// TwinCAT 3 PLC project PLC
// ProgramVersion: 3.1.4024.0
// libraries:
//   Tc2_MC2, * (Beckhoff Automation GmbH)
//   Tc2_MC2_Drive, * (Beckhoff Automation GmbH)
//   Tc2_Standard, * (Beckhoff Automation GmbH)
//   Tc2_System, * (Beckhoff Automation GmbH)
//   Tc3_Module, * (Beckhoff Automation GmbH)
// project tree:
//   GVLs/ GVL.TcGVL
//   / PlcTask.TcTTO
//   POUs/ FB_AxisStMachine.TcPOU (not stored), FB_Axis.TcPOU, FB_AxisStMachineMaster.TcPOU, MAIN.TcPOU
// real-time tasks:
//   TASK PlcTask: cycle T#10ms, priority 20, ADS port 350
// motion (NC):
//   TASK NC-Task 1 SAF: cycle T#2ms, priority 4, ADS port 501
//   TASK NC-Task 1 SVB: cycle T#10ms, priority 8, ADS port 511
//   AXIS Stepper (id 1)
//     General: UnitName=°
//     Dynamic: Acceleration=4263.16, Deceleration=4263.16, Jerk=12789.5
//     Velo: RefSearch=28.42105, RefSync=28.42105, SlowManual=142.10525, FastManual=852.6315, Fast=2842.105, Maximum=2842.11
//     OtherSettings: AllowMotionCmdToSlave=true
//     encoder EncType=4
//       EncPara: ScaleFactorNumerator=360, ScaleFactorDenominator=4096, MaxCount=#x0000ffff
//         Inc: RefSoftSyncMask=#x0000ffff
//         TimeComp: EncDelayCycles=4
//     drive DrvType=24
//       Analog: VeloReferenz=7200, TorqueSetpointScale=10, ScaleFactorActTorque=0.1
//       TimeComp: TaskDelayCycles=1
//     controller CtrType=1
//       CtrPara: PriorControlFactor=1
//         PID: PosKp=50
//         Observer: BandWidth=20
//   AXIS Line1LeftA (id 2)
//     Dynamic: Acceleration=7354.05, Deceleration=7354.05, Jerk=22062.1
//     Velo: RefSearch=49.02699, RefSync=49.02699, SlowManual=245.13495, FastManual=1470.8097, Fast=4902.699, Maximum=4902.7
//     OtherSettings: AllowMotionCmdToSlave=true
//     encoder EncType=19
//       EncPara: ScaleFactorNumerator=60, ScaleFactorDenominator=1048576, MaxCount=#xffffffff
//     drive DrvType=16
//       DrvPara: MaxCount=#xffffffff, DriveControlDWord=#x00020100
//         Analog: VeloReferenz=5392.9689, VeloScale=71.5255737304688, TorqueSetpointScale=10, ScaleFactorActTorque=0.1
//         TimeComp: TaskDelayCycles=1
//     controller CtrType=1
//       CtrPara: PriorControlFactor=1
//         Observer: BandWidth=20
//   AXIS Line2RightB (id 3)
//     Dynamic: Acceleration=7354.05, Deceleration=7354.05, Jerk=22062.1
//     Velo: RefSearch=49.02699, RefSync=49.02699, SlowManual=245.13495, FastManual=1470.8097, Fast=4902.699, Maximum=4902.7
//     OtherSettings: AllowMotionCmdToSlave=true
//     encoder EncType=19
//       EncPara: ScaleFactorNumerator=60, ScaleFactorDenominator=1048576, MaxCount=#xffffffff
//     drive DrvType=16
//       DrvPara: MaxCount=#xffffffff, DriveControlDWord=#x00020100
//         Analog: VeloReferenz=5392.9689, VeloScale=71.5255737304688, TorqueSetpointScale=10, ScaleFactorActTorque=0.1
//         TimeComp: TaskDelayCycles=1
//     controller CtrType=1
//       CtrPara: PriorControlFactor=1
//         Observer: BandWidth=20
//   AXIS RobotMasterVirtualAxe (id 4)
//     OtherSettings: AllowMotionCmdToSlave=true
//     encoder EncType=1
//     drive DrvType=5
//       Analog: TorqueSetpointScale=10, ScaleFactorActTorque=0.1
//       TimeComp: TaskDelayCycles=1
//     controller CtrType=1
//       CtrPara: PriorControlFactor=1
//         Observer: BandWidth=20
// I/O:
//   DEVICE Device 2 (EtherCAT), AmsNetId 172.16.17.50.3.1
//     Term 1 (EK1100) [EK1100 EtherCAT Coupler (2A E-Bus)]
//       Term 2 (EL1004) [EL1004 4Ch. Dig. Input 24V, 3ms]
//       Term 3 (EL2004) [EL2004 4Ch. Dig. Output 24V, 0.5A]
//       Term 4 (EL3062) [EL3062 2Ch. Ana. Input 0-10V]
//       Term 5 (EL7037) [EL7037 1Ch. Stepper motor output stage (24V, 1.5A)]
//         startup 32786:5 := 02 // STM Features Ch.1 / Speed range
//         startup 32785:1 := DE01 // STM Controller Settings Ch.1 / Kp factor (curr.)
//         startup 32785:2 := A200 // STM Controller Settings Ch.1 / Ki factor (curr.)
//         startup 32788:3 := C0010000 // STM Controller Settings 3 Ch.1 / Kp factor (velo.)
//         startup 32788:4 := 8813 // STM Controller Settings 3 Ch.1 / Tn (velo.)
//         startup 32786:8 := 00 // STM Features Ch.1 / Feedback type
//       Term 6 (EL9510) [EL9510 Power supply terminal 10V]
//       Term 9 (EL9011) [EL9011 End Terminal]
//     Term 7 (AX8620-0000-0105) [AX8620-0000-0105]
//       Drive 8 (AX8206-0210-0104) [AX8206-0210-0104 (2Ch. 6A servo axis, safe-motion, multi-FB)]
//         modules: Device, Device, Device, Device, Device, Device, Device, Device, Device, Device, Device (Safety), Device, Device, Device, Device, Device, Device, Device, Device, Device, Device, Device, Device, Device, Device, Device, Device, Device, Device, Device, Device, Line1Left, Line1Left, Line1Left, Line1Left, Line1Left, Line1Left, Line1Left, Line1Left, Line1Left, Line1Left, Line1Left, Line1Left, Line1Left, Line1Left, Line1Left, Line1Left, Line1Left, Line1Left, Line1Left, Line1Left, Line1Left, Line1Left, Line1Left, Line1Left, Line1Left, Line1Left, Line2Right, Line2Right, Line2Right, Line2Right, Line2Right, Line2Right, Line2Right, Line2Right, Line2Right, Line2Right, Line2Right, Line2Right, Line2Right, Line2Right, Line2Right, Line2Right, Line2Right, Line2Right, Line2Right, Line2Right, Line2Right, Line2Right, Line2Right, Line2Right, Line2Right, Line2Right
//         startup 12992:1 := 414D383032312D78427830 // Ch A Motor parameters / Configured motor type
//         startup 24768:0 := FEFF // Ch A Interpolation sub mode select
//         startup 13000:5 := 0200 // Ch A Motor thermal model / Reaction
//         startup 13000:6 := 0000C841 // Ch A Motor thermal model / Partial fraction factor
//         startup 12992:12 := 0000FA45 // Ch A Motor parameters / Motor rated speed
//         startup 12992:13 := C9E5FF3E // Ch A Motor parameters / Motor rated torque
//         startup 24694:0 := F4010000 // Ch A Motor standstill torque
//         startup 24800:0 := D007 // Ch A Positive torque/force limit value
//         startup 24801:0 := D007 // Ch A Negative torque/force limit value
//         startup 12288:6 := 4158383230362D303231302D30303030 // Ch A AxisMain parameters / Configured drive type
//         startup 12867:1 := 9A99593F // Ch A TorqueCtrl parameters / Configured channel rated current
//         startup 12867:2 := 33332340 // Ch A TorqueCtrl parameters / Configured channel peak current
//         startup 12867:7 := 77BE1F40 // Ch A TorqueCtrl parameters / Iuvw max sum
//         startup 24672:0 := 08 // Ch A Modes of operation
//         startup 12864:1 := 0D4D7043 // Ch A TorqueCtrl parameters mappable / Torque control proportional gain q
//         startup 12864:2 := 8A0E7C39 // Ch A TorqueCtrl parameters mappable / Torque control integral action time q
//         startup 12608:1 := 0480D53B // Ch A VeloCtrl parameters mappable / Velocity control proportional gain
//         startup 12608:2 := 6F12033C // Ch A VeloCtrl parameters mappable / Velocity control integral action time
//         startup 12608:3 := 00203246 // Ch A VeloCtrl parameters mappable / Bipolar velocity limit value
//         startup 12992:15 := 0100 // Ch A Motor parameters / Motor temperature sensor connection
//         startup 12611:4 := 0400 // Ch A VeloCtrl observer / Observer type
//         startup 24672:0 := 08 // Ch A Modes of operation
//         startup 12296:2 := 00 // Ch A AxisMain parameters encoder polarity / Primary encoder actual values
//         startup 14016:1 := 414D383032312D78427831 // Ch B Motor parameters / Configured motor type
//         startup 26816:0 := FEFF // Ch B Interpolation sub mode select
//         startup 14024:5 := 0200 // Ch B Motor thermal model / Reaction
//         startup 14024:6 := 0000C841 // Ch B Motor thermal model / Partial fraction factor
//         startup 14016:12 := 0000FA45 // Ch B Motor parameters / Motor rated speed
//         startup 14016:13 := C9E5FF3E // Ch B Motor parameters / Motor rated torque
//         startup 26742:0 := F4010000 // Ch B Motor standstill torque
//         startup 26848:0 := D007 // Ch B Positive torque/force limit value
//         startup 26849:0 := D007 // Ch B Negative torque/force limit value
//         startup 13312:6 := 4158383230362D303231302D30303030 // Ch B AxisMain parameters / Configured drive type
//         startup 13891:1 := 9A99593F // Ch B TorqueCtrl parameters / Configured channel rated current
//         startup 13891:2 := 33332340 // Ch B TorqueCtrl parameters / Configured channel peak current
//         startup 13891:7 := 77BE1F40 // Ch B TorqueCtrl parameters / Iuvw max sum
//         startup 26720:0 := 08 // Ch B Modes of operation
//         startup 13888:1 := 0D4D7043 // Ch B TorqueCtrl parameters mappable / Torque control proportional gain q
//         startup 13888:2 := 8A0E7C39 // Ch B TorqueCtrl parameters mappable / Torque control integral action time q
//         startup 13632:1 := 870B223C // Ch B VeloCtrl parameters mappable / Velocity control proportional gain
//         startup 13632:2 := 6F12033C // Ch B VeloCtrl parameters mappable / Velocity control integral action time
//         startup 13632:3 := 00980546 // Ch B VeloCtrl parameters mappable / Bipolar velocity limit value
//         startup 14016:15 := 0100 // Ch B Motor parameters / Motor temperature sensor connection
//         startup 13635:4 := 0400 // Ch B VeloCtrl observer / Observer type
//         startup 26720:0 := 08 // Ch B Modes of operation
//         startup 13320:2 := 00 // Ch B AxisMain parameters encoder polarity / Primary encoder actual values
// variable links:
//   Device 2 (EtherCAT) <-> Device 2 (EtherCAT)/Term 7 (AX8620-0000-0105)/Drive 8 (AX8206-0210-0104)
//     Term 7 (AX8620-0000-0105)/PSM Controlword for axis/Controlword for axis <-> Device/DeviceMain Outputs/Power supply controlword
//   NC-Task 1 SAF/Axes/Line1LeftA <-> Device 2 (EtherCAT)/Term 7 (AX8620-0000-0105)/Drive 8 (AX8206-0210-0104)
//     Drive/Inputs/In/nDataIn1 <-> Line1Left/Ch A PositionControl Inputs/Ch A Following error actual value
//     Drive/Inputs/In/nDataIn3[0] <-> Line1Left/Ch A TorqueControl Inputs/Ch A Torque/force actual value
//     Drive/Inputs/In/nDcOutputTime <-> InfoData/DcOutputShift
//     Drive/Inputs/In/nState1 <-> Line1Left/Ch A AxisMain Inputs/Ch A Statusword
//     Drive/Inputs/In/nState2 <-> Line1Left/Ch A AxisMain Inputs/Ch A Statusword @bit 8
//     Drive/Inputs/In/nState4 @bit 1 <-> WcState/InputToggle0
//     Drive/Inputs/In/nState4 <-> WcState/WcState0
//     Drive/Outputs/Out/nCtrl1 <-> Line1Left/Ch A AxisMain Outputs/Ch A Controlword
//     Drive/Outputs/Out/nCtrl2 <-> Line1Left/Ch A AxisMain Outputs/Ch A Controlword @bit 8
//     Drive/Outputs/Out/nDataOut1 <-> Line1Left/Ch A Interpolator Outputs/Ch A Target position
//     Drive/Outputs/Out/nDataOut2 <-> Line1Left/Ch A Interpolator Outputs/Ch A Target velocity
//     Enc/Inputs/In/nDataIn1 <-> Line1Left/Ch A AxisMain Inputs/Ch A Position actual value
//     Enc/Inputs/In/nDcInputTime <-> InfoData/DcInputShift
//     Enc/Inputs/In/nState2 @bit 5 <-> Line1Left/Ch A AxisMain Inputs/Position actual value invalid
//     Enc/Inputs/In/nState4 @bit 1 <-> WcState/InputToggle0
//     Enc/Inputs/In/nState4 <-> WcState/WcState0
//   NC-Task 1 SAF/Axes/Line2RightB <-> Device 2 (EtherCAT)/Term 7 (AX8620-0000-0105)/Drive 8 (AX8206-0210-0104)
//     Drive/Inputs/In/nDataIn1 <-> Line2Right/Ch B PositionControl Inputs/Ch B Following error actual value
//     Drive/Inputs/In/nDcOutputTime <-> InfoData/DcOutputShift
//     Drive/Inputs/In/nState1 <-> Line2Right/Ch B AxisMain Inputs/Ch B Statusword
//     Drive/Inputs/In/nState2 <-> Line2Right/Ch B AxisMain Inputs/Ch B Statusword @bit 8
//     Drive/Inputs/In/nState4 @bit 1 <-> WcState/InputToggle0
//     Drive/Inputs/In/nState4 <-> WcState/WcState0
//     Drive/Outputs/Out/nCtrl1 <-> Line2Right/Ch B AxisMain Outputs/Ch B Controlword
//     Drive/Outputs/Out/nCtrl2 <-> Line2Right/Ch B AxisMain Outputs/Ch B Controlword @bit 8
//     Drive/Outputs/Out/nDataOut1 <-> Line2Right/Ch B Interpolator Outputs/Ch B Target position
//     Drive/Outputs/Out/nDataOut2 <-> Line2Right/Ch B Interpolator Outputs/Ch B Target velocity
//     Enc/Inputs/In/nDataIn1 <-> Line2Right/Ch B AxisMain Inputs/Ch B Position actual value
//     Enc/Inputs/In/nDcInputTime <-> InfoData/DcInputShift
//     Enc/Inputs/In/nState2 @bit 5 <-> Line2Right/Ch B AxisMain Inputs/Position actual value invalid
//     Enc/Inputs/In/nState4 @bit 1 <-> WcState/InputToggle0
//     Enc/Inputs/In/nState4 <-> WcState/WcState0
//   NC-Task 1 SAF/Axes/Stepper <-> Device 2 (EtherCAT)/Term 1 (EK1100)/Term 5 (EL7037)
//     Drive/Inputs/In/nState1 @bit 3 <-> STM Status/Status/Error
//     Drive/Inputs/In/nState1 @bit 7 <-> STM Status/Status/Motor stall
//     Drive/Inputs/In/nState1 @bit 5 <-> STM Status/Status/Moving negative
//     Drive/Inputs/In/nState1 @bit 4 <-> STM Status/Status/Moving positive
//     Drive/Inputs/In/nState1 @bit 1 <-> STM Status/Status/Ready
//     Drive/Inputs/In/nState1 <-> STM Status/Status/Ready to enable
//     Drive/Inputs/In/nState1 @bit 6 <-> STM Status/Status/Torque reduced
//     Drive/Inputs/In/nState1 @bit 2 <-> STM Status/Status/Warning
//     Drive/Inputs/In/nState2 @bit 3 <-> STM Status/Status/Digital input 1
//     Drive/Inputs/In/nState2 @bit 4 <-> STM Status/Status/Digital input 2
//     Drive/Inputs/In/nState2 @bit 5 <-> STM Status/Status/Sync error
//     Drive/Inputs/In/nState2 @bit 7 <-> STM Status/Status/TxPDO Toggle
//     Drive/Inputs/In/nState4 @bit 1 <-> WcState/InputToggle
//     Drive/Inputs/In/nState4 <-> WcState/WcState
//     Drive/Outputs/Out/nCtrl1 <-> STM Control/Control/Enable
//     Drive/Outputs/Out/nCtrl1 @bit 2 <-> STM Control/Control/Reduce torque
//     Drive/Outputs/Out/nCtrl1 @bit 1 <-> STM Control/Control/Reset
//     Drive/Outputs/Out/nCtrl2 @bit 3 <-> STM Control/Control/Digital output 1
//     Drive/Outputs/Out/nDataOut2[0] <-> STM Velocity/Velocity
//     Enc/Inputs/In/nDataIn1[0] <-> ENC Status compact/Counter value
//     Enc/Inputs/In/nDataIn2[0] <-> ENC Status compact/Latch value
//     Enc/Inputs/In/nState1 @bit 4 <-> ENC Status compact/Status/Counter overflow
//     Enc/Inputs/In/nState1 @bit 3 <-> ENC Status compact/Status/Counter underflow
//     Enc/Inputs/In/nState1 @bit 7 <-> ENC Status compact/Status/Extrapolation stall
//     Enc/Inputs/In/nState1 <-> ENC Status compact/Status/Latch C valid
//     Enc/Inputs/In/nState1 @bit 1 <-> ENC Status compact/Status/Latch extern valid
//     Enc/Inputs/In/nState1 @bit 2 <-> ENC Status compact/Status/Set counter done
//     Enc/Inputs/In/nState2 @bit 4 <-> ENC Status compact/Status/Status of extern latch
//     Enc/Inputs/In/nState2 <-> ENC Status compact/Status/Status of input A
//     Enc/Inputs/In/nState2 @bit 1 <-> ENC Status compact/Status/Status of input B
//     Enc/Inputs/In/nState2 @bit 2 <-> ENC Status compact/Status/Status of input C
//     Enc/Inputs/In/nState2 @bit 5 <-> ENC Status compact/Status/Sync error
//     Enc/Inputs/In/nState2 @bit 7 <-> ENC Status compact/Status/TxPDO Toggle
//     Enc/Inputs/In/nState4 @bit 1 <-> WcState/InputToggle
//     Enc/Inputs/In/nState4 <-> WcState/WcState
//     Enc/Outputs/Out/nCtrl1 <-> ENC Control compact/Control/Enable latch C
//     Enc/Outputs/Out/nCtrl1 @bit 3 <-> ENC Control compact/Control/Enable latch extern on negative edge
//     Enc/Outputs/Out/nCtrl1 @bit 1 <-> ENC Control compact/Control/Enable latch extern on positive edge
//     Enc/Outputs/Out/nCtrl1 @bit 2 <-> ENC Control compact/Control/Set counter
//     Enc/Outputs/Out/nDataOut1[0] <-> ENC Control compact/Set counter value
//   PLC/PLC Instance <-> Device 2 (EtherCAT)/Term 1 (EK1100)/Term 2 (EL1004)
//     PlcTask Inputs/MAIN.fbAxisStMachine.bCalibCam <-> Channel 4/Input
//     PlcTask Inputs/MAIN.fbAxisStMachine.bDemandStop <-> Channel 2/Input
//     PlcTask Inputs/MAIN.fbAxisStMachine.bDemandVel <-> Channel 1/Input
//   PLC/PLC Instance <-> NC-Task 1 SAF/Axes/Line1LeftA
//     PlcTask Inputs/GVL.Axis_servoA.NcToPlc <-> Outputs/ToPlc
//     PlcTask Outputs/GVL.Axis_servoA.PlcToNc <-> Inputs/FromPlc
//   PLC/PLC Instance <-> NC-Task 1 SAF/Axes/Line2RightB
//     PlcTask Inputs/GVL.Axis_servoB.NcToPlc <-> Outputs/ToPlc
//     PlcTask Outputs/GVL.Axis_servoB.PlcToNc <-> Inputs/FromPlc
//   PLC/PLC Instance <-> NC-Task 1 SAF/Axes/RobotMasterVirtualAxe
//     PlcTask Inputs/GVL.Axis_servoVirtual.NcToPlc <-> Outputs/ToPlc
//     PlcTask Outputs/GVL.Axis_servoVirtual.PlcToNc <-> Inputs/FromPlc
//   PLC/PLC Instance <-> NC-Task 1 SAF/Axes/Stepper
//     PlcTask Inputs/GVL.Axis_servo.NcToPlc <-> Outputs/ToPlc
//     PlcTask Outputs/GVL.Axis_servo.PlcToNc <-> Inputs/FromPlc

CONFIGURATION PLC
    RESOURCE PLC ON TwinCAT3
        TASK PlcTask(INTERVAL := T#10ms, PRIORITY := 20);
        PROGRAM MAIN WITH PlcTask : MAIN;
    END_RESOURCE
END_CONFIGURATION

// ---- GVLs/GVL.TcGVL
{attribute 'qualified_only'}
VAR_GLOBAL
	Axis_servoA : AXIS_REF;
	Axis_servoB : AXIS_REF;
	Axis_servoVirtual : AXIS_REF;
	Axis_servo : AXIS_REF; 
END_VAR

// ---- POUs/MAIN.TcPOU
PROGRAM MAIN
VAR
	myAxisA : FB_Axis;
	myAxisB : FB_Axis;
	myAxisVirtual : FB_Axis;
	myAxisStepper : FB_Axis;
	fbAxisStMachine : FB_AxisStMachine;
END_VAR

//myAxisA(AxisInOut := GVL.Axis_servoA);
//myAxisB(AxisInOut := GVL.Axis_servoB);
//myAxisVirtual(AxisInOut := GVL.Axis_servoVirtual);
//myAxisStepper(AxisInOut := GVL.Axis_servo);

fbAxisStMachine(AxisInOut := GVL.Axis_servoA);

END_PROGRAM

// ---- POUs/FB_Axis.TcPOU
FUNCTION_BLOCK FB_Axis
VAR_INPUT
END_VAR
VAR_OUTPUT
END_VAR
VAR_IN_OUT
	AxisInOut : AXIS_REF;//AXIS_REF contains input and output
END_VAR
VAR
	fbPower : MC_Power;
	fbMoveAbs : MC_MoveAbsolute;
	fTarget	: LREAL := 720;
	fVelocity : LREAL := 360;
	
	errId : UDINT;
	bBusy,bError, bMove, bDone : BOOL;
END_VAR

AxisInOut.ReadStatus();//must be always called each cycle

fbPower(
	Axis:= AxisInOut, 
	Enable:= TRUE, 
	Enable_Positive:= TRUE, 
	Enable_Negative:= TRUE, 
	Override:= 100, 
	Busy=>bBusy , 
	Error=> bError, 
	ErrorID=> errId);
	
fbMoveAbs(
	Axis:= AxisInOut, 
	Execute:= bMove, 
	Position:= fTarget, 
	Velocity:= fVelocity,  
	Done=> bDone, 
	Busy=>bBusy, 
	Error=>bError, 
	ErrorID=> errId);

END_FUNCTION_BLOCK

// ---- POUs/FB_AxisStMachineMaster.TcPOU
FUNCTION_BLOCK FB_AxisStMachineMaster
VAR_IN_OUT
	AxisInOut : AXIS_REF;//AXIS_REF contains input and output
END_VAR
VAR
	nStep : UINT := 10;
	
	fbPower : MC_Power;
		
	errId : UDINT;
	bBusy, bError, bMoveAbs, bMoveVel, bDone, bPower, bReset, bResetDone,bVelocity, bInVelocity, MoveAbsbDone, bDoneHalt, bAborted,bHalt,bHomingDone : BOOL;

	bDemandStop,bDemandVel  AT%I* : BOOL;
	
	fbMoveAbs : MC_MoveAbsolute;
	fTarget	: LREAL := 720;
	fVelocity : LREAL := 36;
	fVelocityInfinite : LREAL := 360;
	fbReset : MC_Reset;//remove error in the NC only for AX8000 but not for AX5000
	fbVelocity : MC_MoveVelocity;
	fbHalt : MC_HALT;
	fbHome : MC_Home;
	bCalibCam AT%I* : BOOL;
	bHome : BOOL;
END_VAR

RunFBs();

CASE nStep OF
	0 : //Idle
		;
	10:
		bPower := TRUE;
		nStep := 15;
	15:
		IF AxisInOut.Status.Error THEN //really at the level of NC
			nStep := 20;
		ELSE
			nstep := 40;
		END_IF
	20:
		bReset := TRUE;
		nstep := 30;	
	30:
		IF bResetDone THEN
			bReset := FALSE;
			nStep := 40;
		END_IF
	40:
		IF fbPower.Status THEN
			bHome := TRUE;
			nStep := 45;
		END_IF
	45:
		IF bHomingDone THEN
			bHome := FALSE;
			nStep := 50;
		END_IF 
	50:
		bMoveAbs := TRUE;
		fTarget	 := 36;//gradi
		fVelocity := 36;
		nstep := 60;
	60:
		IF MoveAbsbDone THEN
			bMoveAbs := FALSE;
			nStep := 65;
		END_IF
	65:
		IF bDemandVel THEN
			nStep := 70;
		END_IF
	70:
		bMoveVel := TRUE;
		fVelocityInfinite := 1440;
		nStep := 80;
	80:
		IF bDemandStop THEN
			bMoveVel := FALSE;
			nStep := 90;
		END_IF
	90:
		bHalt := TRUE;
		nStep := 100;
	
	100:
		IF fbHalt.Done THEN
			bHalt := FALSE;
			nStep := 0;
		END_IF
	ELSE
		;
END_CASE

METHOD RunFBs : BOOL
fbPower(
	Axis:= AxisInOut, 
	Enable:= bPower, 
	Enable_Positive:= TRUE, 
	Enable_Negative:= TRUE, 
	Override:= 100, 
	Busy=>bBusy , 
	Error=>bError, 
	ErrorID=> errId);

fbMoveAbs(
	Axis:= AxisInOut, 
	Execute:= bMoveAbs, 
	Position:= fTarget, 
	Velocity:= fVelocity,  
	Done=> MoveAbsbDone, 
	Busy=>bBusy, 
	Error=>bError, 
	ErrorID=> errId);

fbReset(
	Axis:= AxisInOut, 
	Execute:= bReset, 
	Done=> bResetDone,
	Busy=> bBusy, 
	Error=>bError, 
	ErrorID=>errId);
	
fbVelocity(
	Axis:= AxisInOut, 
	Execute:= bMoveVel, 
	Velocity:= fVelocityInfinite, 
	InVelocity=> bInVelocity, 
	Busy=> bBusy, 
	Error=>bError, 
	ErrorID=>errId);

fbHalt(
	Axis:= AxisInOut, 
	Execute:= bHalt, 
	Done=> bDoneHalt, 
	Busy=> bBusy, 
	CommandAborted=> bAborted, 
	Error=> bError, 
	ErrorID=>errId);

	//without giving special values to the parameters NC parameters are used
fbHome(
	Axis:= AxisInOut, 
	Execute:= bHome, 
	Position:= , 
	HomingMode:= , 
	BufferMode:= , 
	Options:= , 
	bCalibrationCam:= bCalibCam, 
	Done=> bHomingDone, 
	Busy=> , 
	Active=> , 
	CommandAborted=> , 
	Error=> , 
	ErrorID=> );
END_METHOD

END_FUNCTION_BLOCK
